# EPICS autosave request: iocBoot/iocpmcvtest/auto_positions.req
file motor_positions.req P=MLL:,M=pmcv1
file motor_positions.req P=MLL:,M=pmcv2
file motor_positions.req P=MLL:,M=pmcv3
